cmd.FB_Build(
	rDoExtending := rDoExtending,
	rDoRetracting := rDoRetracting,
	rDiAtExtendedPosition := rDiAtExtendedPosition,
	commandTimeout := T#5S
);

(* stored: Version 1.1.0.1
   POU P: Id {b} *)
